PROGRAM Cell_SafetyMapping
VAR

END_VAR

END_PROGRAM

(* stored: Version 1.1.0.1, ProductVersion 3.1.4022.11
   POU Cell_SafetyMapping: Id {80ae55d1-70f2-4389-b7f8-ac53585c12b2}, SpecialFunc None *)
